// TIA Portal V19 export
DATA_BLOCK "Gripper_MeasuInput"   // DB156, Motion_DB
// stored: InstanceOfName TO_MeasuringInput, OfSystemLibElement TO_MeasuringInput, OfSystemLibVersion 8.0
TO_MeasuringInput   // technology object, version 8.0
// stored: Connection Interface MeasuringInput, InputAddress 2957
   // // inherited from TO_Object
   // VAR
   //    Status { ExternalWritable := 'False'} : DInt;
   //    InputState { ExternalWritable := 'False'} : Bool;
   //    Parameter { S7_SetPoint := 'True'} : TO_MeasuringInput_Struct_Parameter;
   //    Interface { ExternalWritable := 'False'; S7_SetPoint := 'True'} : TO_MeasuringInput_Struct_Interface;
   //    MeasuredValues { ExternalWritable := 'False'; S7_SetPoint := 'True'} : TO_MeasuringInput_Struct_MeasuredValues;
   //    Units { ExternalWritable := 'False'; S7_SetPoint := 'True'} : TO_MeasuringInput_Struct_Units;
   //    StatusWord { ExternalWritable := 'False'} : DWord;
   //    ErrorWord { ExternalWritable := 'False'} : DWord;
   //    ErrorDetail { ExternalWritable := 'False'; S7_SetPoint := 'True'} : TO_Struct_ErrorDetail;
   //    WarningWord { ExternalWritable := 'False'} : DWord;
   // END_VAR
BEGIN
   Parameter.MeasuringRangeActivationTime := 0.5;
   Interface.Address.RID := 16#2000001;
   Interface.Address.AREA := 16#81;
   Interface.Address.OFFSET := 2957;
END_DATA_BLOCK
